// TIA Portal V17 export
// export: Created 2022-01-22T12:57:25.3275354Z, ExportSetting WithDefaults, DisplayName Totally Integrated Automation Portal, DisplayVersion V17 Update 2, DisplayName TIA Portal Openness, DisplayVersion V17 Update 2, DisplayName TIA Portal Version Control Interface, DisplayVersion V17, DisplayName SINAMICS Startdrive Advanced, DisplayVersion V17, DisplayName SINAMICS Startdrive G130, G150, S120, S150, SINAMICS MV, S210, DisplayVersion V17, DisplayName SINAMICS Startdrive G110M, G120, G120C, G120D, G120P, G115D, DisplayVersion V17, DisplayName STEP 7 Professional, DisplayVersion V17 Update 2, DisplayName STEP 7 Safety, DisplayVersion V17, DisplayName WinCC UA Professional, DisplayVersion V17 Update 2, DisplayName WinCC Unified Calendar, DisplayVersion V17, DisplayName WinCC Unified LineCoordination, DisplayVersion V17, DisplayName WinCC Unified Performance Insight, DisplayVersion V17, DisplayName WinCC Unified Sequence, DisplayVersion V17, DisplayName SIMATIC Visualization Architect, DisplayVersion V17
FUNCTION_BLOCK "fbTemplateOP"   // FB1, FBD
{ S7_Optimized_Access := 'TRUE' }
VERSION : 0.1
// stored: AutoNumber true, IsIECCheckEnabled false, IsRetainMemResEnabled false, MemoryReserve 100, SetENOAutomatically false, UDAEnableTagReadback false
   VAR
      State { S7_SetPoint := 'True'} : Program_Alarm;
   END_VAR
BEGIN
END_FUNCTION_BLOCK
